// TIA Portal V17 export
// export: Created 2025-03-07T09:18:15.2126979Z, ExportSetting WithDefaults, DisplayName Totally Integrated Automation Portal, DisplayVersion V17 Update 8, DisplayName TIA Portal Openness, DisplayVersion V17 Update 8, DisplayName TIA Portal Version Control Interface, DisplayVersion V17, DisplayName SINAMICS Startdrive Advanced, DisplayVersion V17 SP2, DisplayName SINAMICS Startdrive G110M, G120, G120C, G120D, G120P, G115D, DisplayVersion V17 SP2, DisplayName SINAMICS Startdrive G130, G150, S120, S150, SINAMICS MV, S210, DisplayVersion V17 SP2, DisplayName STEP 7 Professional, DisplayVersion V17 Update 8, DisplayName SINUMERIK ONE STEP 7 Toolbox, DisplayVersion V17 Update 12, DisplayName SINUMERIK 840D sl STEP 7 Toolbox, DisplayVersion V17 Update 12, DisplayName STEP 7 Safety, DisplayVersion V17 Update 6, DisplayName WinCC Advanced, DisplayVersion V17 Update 8
FUNCTION "FC1300_UNIT_03_SEQUENCES" : Void   // FC1300, LAD
{ S7_Optimized_Access := 'FALSE' }
AUTHOR : ETXETAR
VERSION : 1.0
// stored: AutoNumber false, IsIECCheckEnabled false, SetENOAutomatically false, UDAEnableTagReadback false
BEGIN

REGION Network 1: CALL FC1203 PART CYCLE UNIT 01 CLADDING
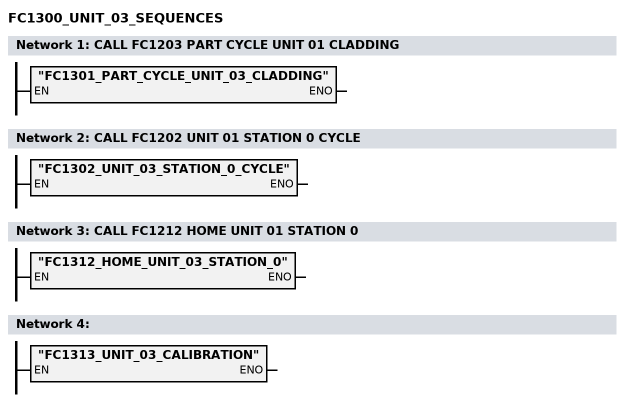
   RUNG wire#powerrail
      "FC1301_PART_CYCLE_UNIT_03_CLADDING"()
   END_RUNG
   // the same network as SCL:
   "FC1301_PART_CYCLE_UNIT_03_CLADDING"();
END_REGION

REGION Network 2: CALL FC1202 UNIT 01 STATION 0 CYCLE
   RUNG wire#powerrail
      "FC1302_UNIT_03_STATION_0_CYCLE"()
   END_RUNG
   // the same network as SCL:
   "FC1302_UNIT_03_STATION_0_CYCLE"();
END_REGION

REGION Network 3: CALL FC1212 HOME UNIT 01 STATION 0
   RUNG wire#powerrail
      "FC1312_HOME_UNIT_03_STATION_0"()
   END_RUNG
   // the same network as SCL:
   "FC1312_HOME_UNIT_03_STATION_0"();
END_REGION

REGION Network 4
   RUNG wire#powerrail
      "FC1313_UNIT_03_CALIBRATION"()
   END_RUNG
   // the same network as SCL:
   "FC1313_UNIT_03_CALIBRATION"();
END_REGION
END_FUNCTION
